SUBAPPLICATION Uebung_006a2b (* 2x SR und T-Flip-Flop mit IX *)
  (* Standard: 61499-2; Description: Copyright (c) 2023 Meisterschulen am Ostbahnhof This program and the accompanying materials are made available under the terms of the Eclipse Public License 2.0 which is available at https://www.eclipse.org/legal/epl-2.0/ SPDX-License-Identifier: EPL-2.0 *)
  (* Version 1.0, 2026-01-13, Franz Höpfinger, Meisterschulen am Ostbahnhof, initial API and implementation and/or initial documentation *)
  PACKAGE Uebungen;
  IMPORT logiBUS::io::DI::logiBUS_DI::Input_I1;
  IMPORT logiBUS::io::DI::logiBUS_DI::Input_I2;
  IMPORT logiBUS::io::DI::logiBUS_DI::Input_I3;
  IMPORT logiBUS::io::DQ::logiBUS_DO::Output_Q1;
  IMPORT logiBUS::io::DQ::logiBUS_DO::Output_Q2;
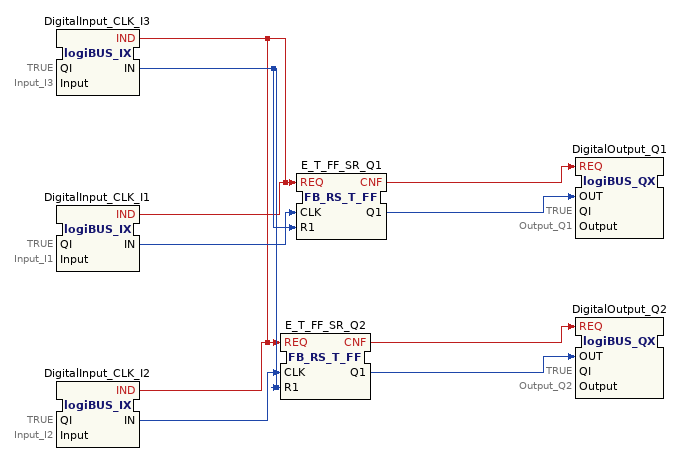
  (* Hausmeister-Aus (alles Aus mit einem Druck) *)
  FBS
    DigitalOutput_Q1 : logiBUS::io::DQ::logiBUS_QX(QI := TRUE, Output := Output_Q1);
    DigitalInput_CLK_I1 : logiBUS::io::DI::logiBUS_IX(QI := TRUE, Input := Input_I1);
    DigitalInput_CLK_I2 : logiBUS::io::DI::logiBUS_IX(QI := TRUE, Input := Input_I2);
    E_T_FF_SR_Q1 : logiBUS::bistableElements::FB_RS_T_FF;
    DigitalInput_CLK_I3 : logiBUS::io::DI::logiBUS_IX(QI := TRUE, Input := Input_I3);
    E_T_FF_SR_Q2 : logiBUS::bistableElements::FB_RS_T_FF;
    DigitalOutput_Q2 : logiBUS::io::DQ::logiBUS_QX(QI := TRUE, Output := Output_Q2);
  END_FBS
  EVENT_CONNECTIONS
    DigitalInput_CLK_I1.IND TO E_T_FF_SR_Q1.REQ;
    DigitalInput_CLK_I2.IND TO E_T_FF_SR_Q2.REQ;
    DigitalInput_CLK_I3.IND TO E_T_FF_SR_Q1.REQ;
    DigitalInput_CLK_I3.IND TO E_T_FF_SR_Q2.REQ;
    E_T_FF_SR_Q1.CNF TO DigitalOutput_Q1.REQ;
    E_T_FF_SR_Q2.CNF TO DigitalOutput_Q2.REQ;
  END_CONNECTIONS
  DATA_CONNECTIONS
    DigitalInput_CLK_I1.IN TO E_T_FF_SR_Q1.CLK;
    DigitalInput_CLK_I2.IN TO E_T_FF_SR_Q2.CLK;
    DigitalInput_CLK_I3.IN TO E_T_FF_SR_Q1.R1;
    DigitalInput_CLK_I3.IN TO E_T_FF_SR_Q2.R1;
    E_T_FF_SR_Q1.Q1 TO DigitalOutput_Q1.OUT;
    E_T_FF_SR_Q2.Q1 TO DigitalOutput_Q2.OUT;
  END_CONNECTIONS
END_SUBAPPLICATION
